INTERFACE I_DigitalInput EXTENDS I_DigitalDevice

PROPERTY EnableForce : BOOL
GET
END_GET
SET
END_SET
END_PROPERTY

PROPERTY FallingTrigger : BOOL
GET
END_GET
END_PROPERTY

PROPERTY In : BOOL
GET
END_GET
END_PROPERTY

METHOD MR_ResetForceValue
END_METHOD

METHOD MR_SetForceValue
END_METHOD

PROPERTY RisingTrigger : BOOL
GET
END_GET
END_PROPERTY

END_INTERFACE

(* stored: Version 1.1.0.1, ProductVersion 3.1.4024.9
   Itf I_DigitalInput: Id {598e54c6-5126-4b16-91f1-a31578c62fc9}
   Property EnableForce: Id {19756f5f-eb61-4f19-a512-86e5f58d5561}
   Get Get: Id {f8926b77-5eca-47f4-95c7-382a953a9864}
   Set Set: Id {e0fd76b2-005b-49a3-b540-0270ba9359c1}
   Property FallingTrigger: Id {b6cc4d2d-0910-4216-8ca8-9708e2f2b075}
   Get Get: Id {2d5e2cc6-5072-4c10-939f-aa8c59a1e76a}
   Property In: Id {f00b1dab-047f-4bf8-a08e-17b87ee2dc8d}
   Get Get: Id {f44289c4-135f-4aa9-8640-a2de0f7ee5a6}
   Method MR_ResetForceValue: Id {ffd57104-d619-4d6c-8e26-1dcae544bbe2}
   Method MR_SetForceValue: Id {c955e1da-884d-4b5a-b167-be532b077564}
   Property RisingTrigger: Id {73be4545-7b24-4cbb-ad2c-0dc8d5327a86}
   Get Get: Id {9c56e293-c6a1-4a24-90e6-ddd8b700564c} *)
